{attribute 'GeneratedUsingTerminal: EL1258-0000-0016'}
{attribute addProperty BoxType "EL1258-0000-0016"}
{attribute addProperty Id "MTI_Inputs_10x_Channel_1AT %I*MTI_Inputs_10x_Channel_C3ED30FD56MTI_Inputs_10x_Channel_2AT %I*MTI_Inputs_10x_Channel_C3ED30FD56MTI_Inputs_10x_Channel_3AT %I*MTI_Inputs_10x_Channel_C3ED30FD56MTI_Inputs_10x_Channel_4AT %I*MTI_Inputs_10x_Channel_C3ED30FD56MTI_Inputs_10x_Channel_5AT %I*MTI_Inputs_10x_Channel_C3ED30FD56MTI_Inputs_10x_Channel_6AT %I*MTI_Inputs_10x_Channel_C3ED30FD56MTI_Inputs_10x_Channel_7AT %I*MTI_Inputs_10x_Channel_C3ED30FD56MTI_Inputs_10x_Channel_8AT %I*MTI_Inputs_10x_Channel_C3ED30FD56MTI_Outputs_Channel_1AT %Q*MTI_Outputs_Channel_0F1028A12MTI_Outputs_Channel_2AT %Q*MTI_Outputs_Channel_0F1028A12MTI_Outputs_Channel_3AT %Q*MTI_Outputs_Channel_0F1028A12MTI_Outputs_Channel_4AT %Q*MTI_Outputs_Channel_0F1028A12MTI_Outputs_Channel_5AT %Q*MTI_Outputs_Channel_0F1028A12MTI_Outputs_Channel_6AT %Q*MTI_Outputs_Channel_0F1028A12MTI_Outputs_Channel_7AT %Q*MTI_Outputs_Channel_0F1028A12MTI_Outputs_Channel_8AT %Q*MTI_Outputs_Channel_0F1028A12WcStateAT %I*WcState_9091E0EB2InfoDataAT %I*InfoData_1088C70510"}
{attribute addProperty CRC "4201081730"}
{attribute addProperty Size "476"}
TYPE EL1258_FA676B82 EXTENDS EtcSlaveTerminalBase_947E5A46 :
STRUCT
	{attribute addProperty Name "MTI_Inputs_10x_Channel_1"}
	MTI_Inputs_10x_Channel_1 : MTI_Inputs_10x_Channel_C3ED30FD;
	{attribute addProperty Name "MTI_Inputs_10x_Channel_2"}
	MTI_Inputs_10x_Channel_2 : MTI_Inputs_10x_Channel_C3ED30FD;
	{attribute addProperty Name "MTI_Inputs_10x_Channel_3"}
	MTI_Inputs_10x_Channel_3 : MTI_Inputs_10x_Channel_C3ED30FD;
	{attribute addProperty Name "MTI_Inputs_10x_Channel_4"}
	MTI_Inputs_10x_Channel_4 : MTI_Inputs_10x_Channel_C3ED30FD;
	{attribute addProperty Name "MTI_Inputs_10x_Channel_5"}
	MTI_Inputs_10x_Channel_5 : MTI_Inputs_10x_Channel_C3ED30FD;
	{attribute addProperty Name "MTI_Inputs_10x_Channel_6"}
	MTI_Inputs_10x_Channel_6 : MTI_Inputs_10x_Channel_C3ED30FD;
	{attribute addProperty Name "MTI_Inputs_10x_Channel_7"}
	MTI_Inputs_10x_Channel_7 : MTI_Inputs_10x_Channel_C3ED30FD;
	{attribute addProperty Name "MTI_Inputs_10x_Channel_8"}
	MTI_Inputs_10x_Channel_8 : MTI_Inputs_10x_Channel_C3ED30FD;
	{attribute addProperty Name "MTI_Outputs_Channel_1"}
	MTI_Outputs_Channel_1 : MTI_Outputs_Channel_0F1028A1;
	{attribute addProperty Name "MTI_Outputs_Channel_2"}
	MTI_Outputs_Channel_2 : MTI_Outputs_Channel_0F1028A1;
	{attribute addProperty Name "MTI_Outputs_Channel_3"}
	MTI_Outputs_Channel_3 : MTI_Outputs_Channel_0F1028A1;
	{attribute addProperty Name "MTI_Outputs_Channel_4"}
	MTI_Outputs_Channel_4 : MTI_Outputs_Channel_0F1028A1;
	{attribute addProperty Name "MTI_Outputs_Channel_5"}
	MTI_Outputs_Channel_5 : MTI_Outputs_Channel_0F1028A1;
	{attribute addProperty Name "MTI_Outputs_Channel_6"}
	MTI_Outputs_Channel_6 : MTI_Outputs_Channel_0F1028A1;
	{attribute addProperty Name "MTI_Outputs_Channel_7"}
	MTI_Outputs_Channel_7 : MTI_Outputs_Channel_0F1028A1;
	{attribute addProperty Name "MTI_Outputs_Channel_8"}
	MTI_Outputs_Channel_8 : MTI_Outputs_Channel_0F1028A1;
	{attribute addProperty Name "WcState"}
	WcState : WcState_9091E0EB;
	{attribute addProperty Name "InfoData"}
	InfoData : InfoData_1088C705;
END_STRUCT
END_TYPE

(* stored: Version 1.2.0.0, ProductVersion 3.1.4024.9
   DUT EL1258_FA676B82: Id {bf226c53-db61-496a-a829-8440917ced62} *)
